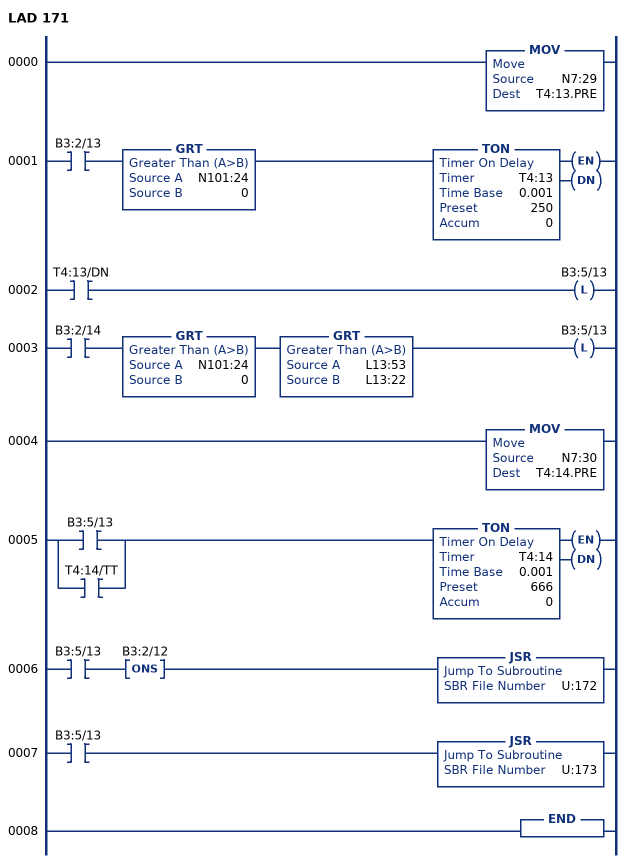
% Rung: 0 %
SOR MOV N7:29 T4:13.PRE EOR
% Rung: 1 %
SOR XIC B3:2/13 GRT N101:24 0 TON T4:13 0.001 250 0 EOR
% Rung: 2 %
SOR XIC T4:13/DN OTL B3:5/13 EOR
% Rung: 3 %
SOR XIC B3:2/14 GRT N101:24 0 GRT L13:53 L13:22 OTL B3:5/13 EOR
% Rung: 4 %
SOR MOV N7:30 T4:14.PRE EOR
% Rung: 5 %
SOR BST XIC B3:5/13 NXB XIC T4:14/TT BND TON T4:14 0.001 666 0 EOR
% Rung: 6 %
SOR XIC B3:5/13 ONS B3:2/12 JSR U:172 EOR
% Rung: 7 %
SOR XIC B3:5/13 JSR U:173 EOR
% Rung: 8 %
SOR END EOR

LADDER 172
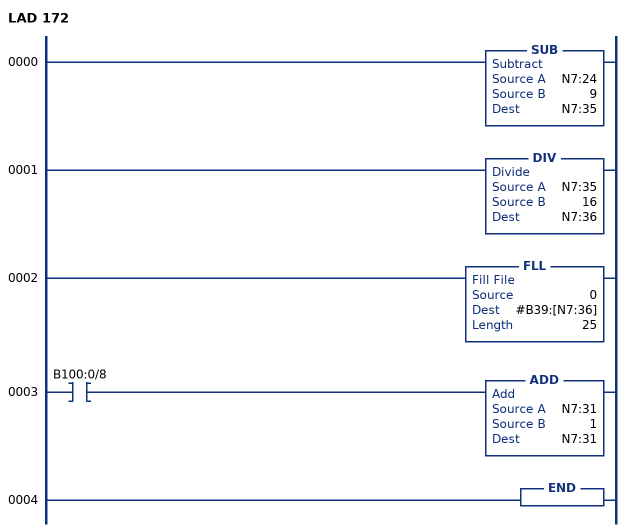
% Rung: 0 %
SOR SUB N7:24 9 N7:35 EOR
% Rung: 1 %
SOR DIV N7:35 16 N7:36 EOR
% Rung: 2 %
SOR FLL 0 #B39:[N7:36] 25 EOR
% Rung: 3 %
SOR XIC B100:0/8 ADD N7:31 1 N7:31 EOR
% Rung: 4 %
SOR END EOR

LADDER 173
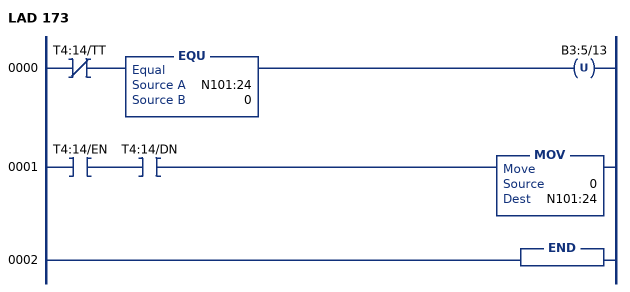
% Rung: 0 %
SOR XIO T4:14/TT EQU N101:24 0 OTU B3:5/13 EOR
% Rung: 1 %
SOR XIC T4:14/EN XIC T4:14/DN MOV 0 N101:24 EOR
% Rung: 2 %
SOR END EOR

LADDER 174
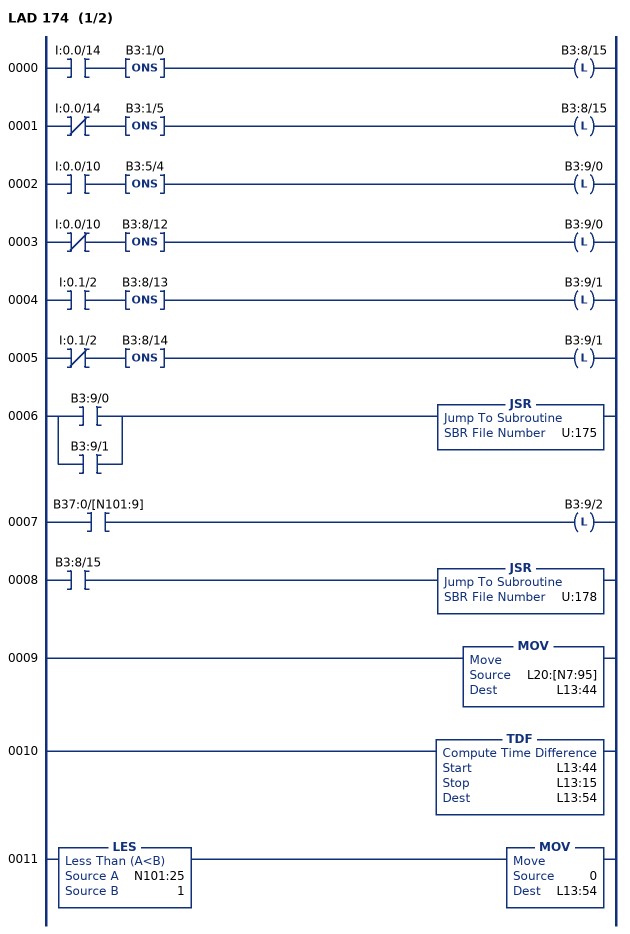
% Rung: 0 %
SOR XIC I:0.0/14 ONS B3:1/0 OTL B3:8/15 EOR
% Rung: 1 %
SOR XIO I:0.0/14 ONS B3:1/5 OTL B3:8/15 EOR
% Rung: 2 %
SOR XIC I:0.0/10 ONS B3:5/4 OTL B3:9/0 EOR
% Rung: 3 %
SOR XIO I:0.0/10 ONS B3:8/12 OTL B3:9/0 EOR
% Rung: 4 %
SOR XIC I:0.1/2 ONS B3:8/13 OTL B3:9/1 EOR
% Rung: 5 %
SOR XIO I:0.1/2 ONS B3:8/14 OTL B3:9/1 EOR
% Rung: 6 %
SOR BST XIC B3:9/0 NXB XIC B3:9/1 BND JSR U:175 EOR
% Rung: 7 %
SOR XIC B37:0/[N101:9] OTL B3:9/2 EOR
% Rung: 8 %
SOR XIC B3:8/15 JSR U:178 EOR
% Rung: 9 %
SOR MOV L20:[N7:95] L13:44 EOR
% Rung: 10 %
SOR TDF L13:44 L13:15 L13:54 EOR
% Rung: 11 %
SOR LES N101:25 1 MOV 0 L13:54 EOR

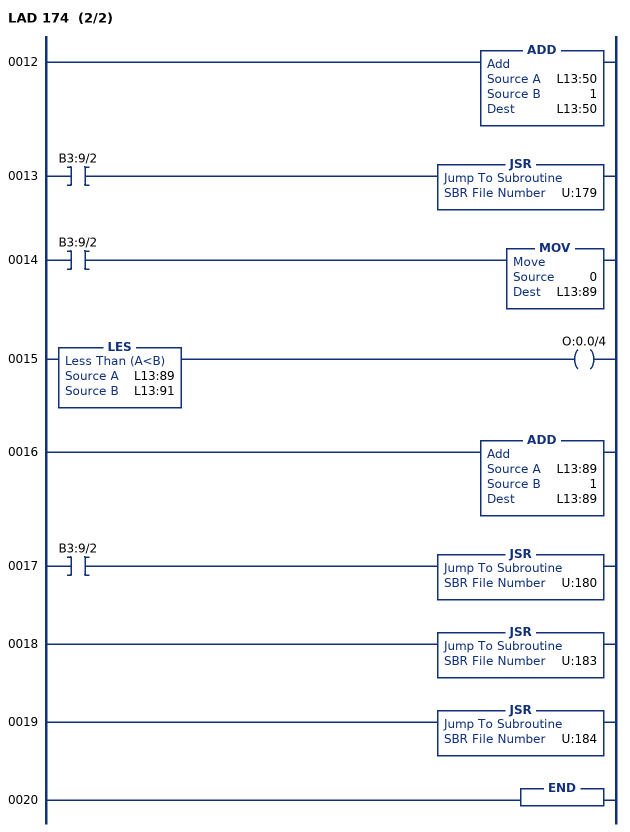
% Rung: 12 %
SOR ADD L13:50 1 L13:50 EOR
% Rung: 13 %
SOR XIC B3:9/2 JSR U:179 EOR
% Rung: 14 %
SOR XIC B3:9/2 MOV 0 L13:89 EOR
% Rung: 15 %
SOR LES L13:89 L13:91 OTE O:0.0/4 EOR
% Rung: 16 %
SOR ADD L13:89 1 L13:89 EOR
% Rung: 17 %
SOR XIC B3:9/2 JSR U:180 EOR
% Rung: 18 %
SOR JSR U:183 EOR
% Rung: 19 %
SOR JSR U:184 EOR
% Rung: 20 %
SOR END EOR

LADDER 175
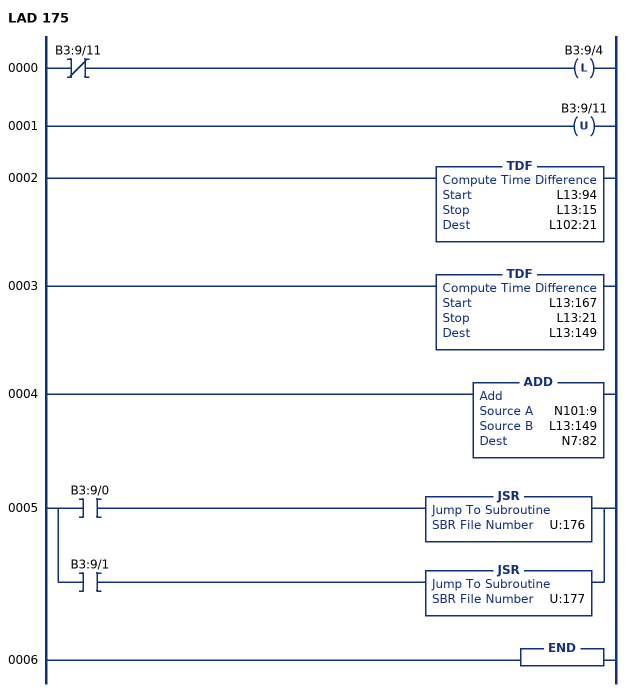
% Rung: 0 %
SOR XIO B3:9/11 OTL B3:9/4 EOR
% Rung: 1 %
SOR OTU B3:9/11 EOR
% Rung: 2 %
SOR TDF L13:94 L13:15 L102:21 EOR
% Rung: 3 %
SOR TDF L13:167 L13:21 L13:149 EOR
% Rung: 4 %
SOR ADD N101:9 L13:149 N7:82 EOR
% Rung: 5 %
SOR BST XIC B3:9/0 JSR U:176 NXB XIC B3:9/1 JSR U:177 BND EOR
% Rung: 6 %
SOR END EOR

LADDER 176
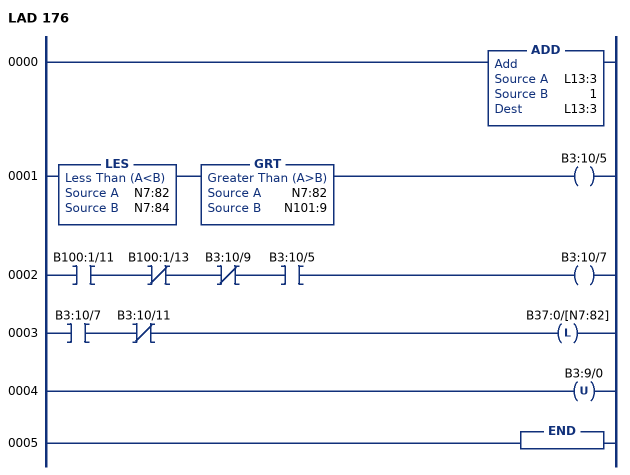
% Rung: 0 %
SOR ADD L13:3 1 L13:3 EOR
% Rung: 1 %
SOR LES N7:82 N7:84 GRT N7:82 N101:9 OTE B3:10/5 EOR
% Rung: 2 %
SOR XIC B100:1/11 XIO B100:1/13 XIO B3:10/9 XIC B3:10/5 OTE B3:10/7 EOR
% Rung: 3 %
SOR XIC B3:10/7 XIO B3:10/11 OTL B37:0/[N7:82] EOR
% Rung: 4 %
SOR OTU B3:9/0 EOR
% Rung: 5 %
SOR END EOR

LADDER 177
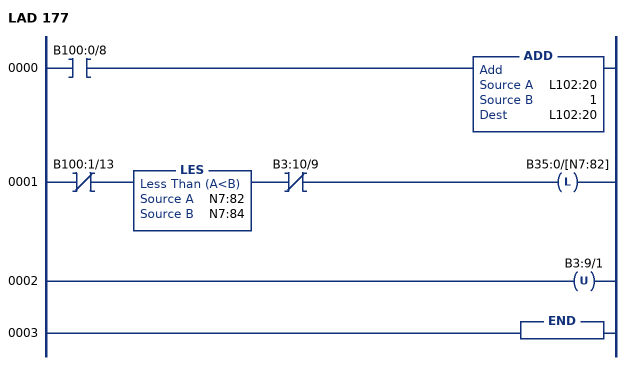
% Rung: 0 %
SOR XIC B100:0/8 ADD L102:20 1 L102:20 EOR
% Rung: 1 %
SOR XIO B100:1/13 LES N7:82 N7:84 XIO B3:10/9 OTL B35:0/[N7:82] EOR
% Rung: 2 %
SOR OTU B3:9/1 EOR
% Rung: 3 %
SOR END EOR

LADDER 178
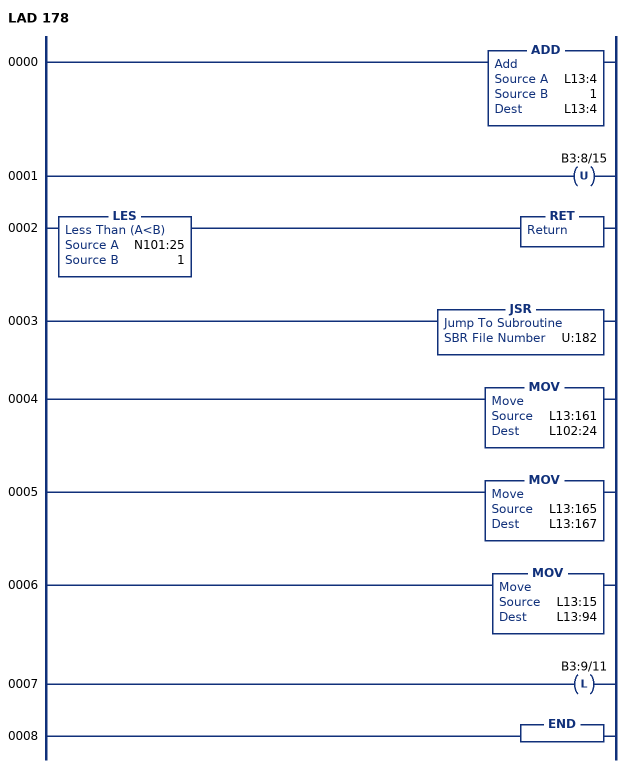
% Rung: 0 %
SOR ADD L13:4 1 L13:4 EOR
% Rung: 1 %
SOR OTU B3:8/15 EOR
% Rung: 2 %
SOR LES N101:25 1 RET EOR
% Rung: 3 %
SOR JSR U:182 EOR
% Rung: 4 %
SOR MOV L13:161 L102:24 EOR
% Rung: 5 %
SOR MOV L13:165 L13:167 EOR
% Rung: 6 %
SOR MOV L13:15 L13:94 EOR
% Rung: 7 %
SOR OTL B3:9/11 EOR
% Rung: 8 %
SOR END EOR

LADDER 179
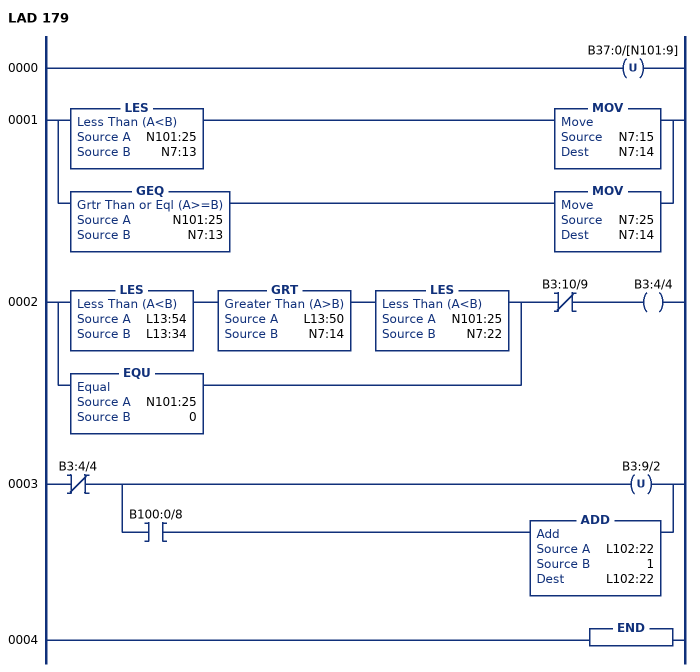
% Rung: 0 %
SOR OTU B37:0/[N101:9] EOR
% Rung: 1 %
SOR BST LES N101:25 N7:13 MOV N7:15 N7:14 NXB GEQ N101:25 N7:13 MOV N7:25 N7:14 BND EOR
% Rung: 2 %
SOR BST LES L13:54 L13:34 GRT L13:50 N7:14 LES N101:25 N7:22 NXB EQU N101:25 0 BND XIO B3:10/9 OTE B3:4/4 EOR
% Rung: 3 %
SOR XIO B3:4/4 BST OTU B3:9/2 NXB XIC B100:0/8 ADD L102:22 1 L102:22 BND EOR
% Rung: 4 %
SOR END EOR

LADDER 180
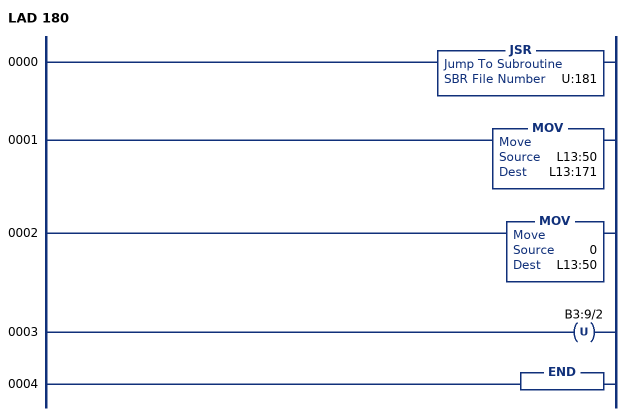
% Rung: 0 %
SOR JSR U:181 EOR
% Rung: 1 %
SOR MOV L13:50 L13:171 EOR
% Rung: 2 %
SOR MOV 0 L13:50 EOR
% Rung: 3 %
SOR OTU B3:9/2 EOR
% Rung: 4 %
SOR END EOR

LADDER 181
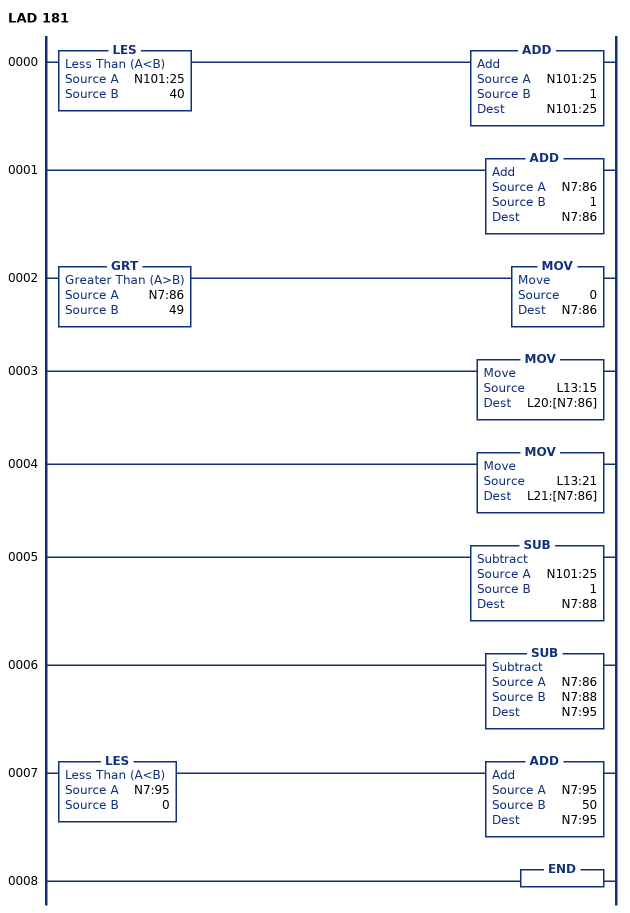
% Rung: 0 %
SOR LES N101:25 40 ADD N101:25 1 N101:25 EOR
% Rung: 1 %
SOR ADD N7:86 1 N7:86 EOR
% Rung: 2 %
SOR GRT N7:86 49 MOV 0 N7:86 EOR
% Rung: 3 %
SOR MOV L13:15 L20:[N7:86] EOR
% Rung: 4 %
SOR MOV L13:21 L21:[N7:86] EOR
% Rung: 5 %
SOR SUB N101:25 1 N7:88 EOR
% Rung: 6 %
SOR SUB N7:86 N7:88 N7:95 EOR
% Rung: 7 %
SOR LES N7:95 0 ADD N7:95 50 N7:95 EOR
% Rung: 8 %
SOR END EOR

LADDER 182
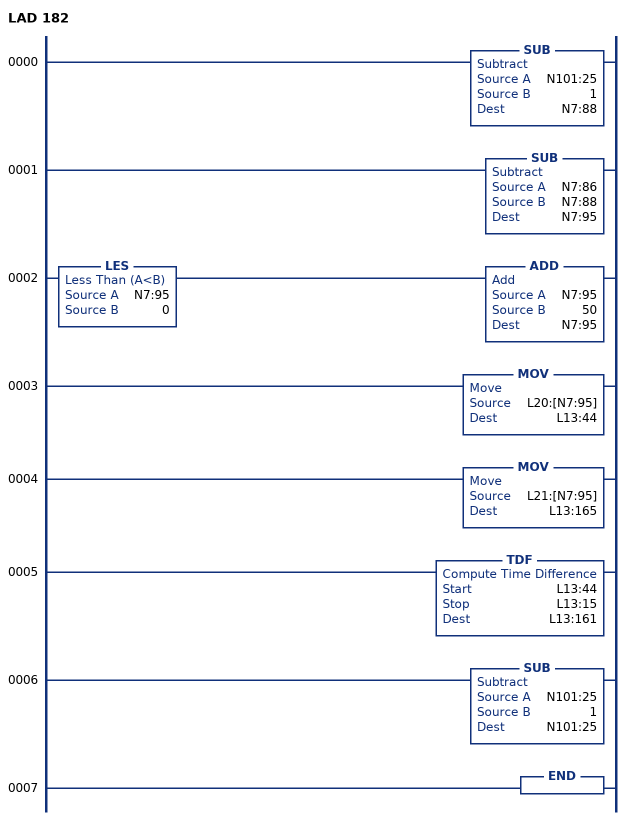
% Rung: 0 %
SOR SUB N101:25 1 N7:88 EOR
% Rung: 1 %
SOR SUB N7:86 N7:88 N7:95 EOR
% Rung: 2 %
SOR LES N7:95 0 ADD N7:95 50 N7:95 EOR
% Rung: 3 %
SOR MOV L20:[N7:95] L13:44 EOR
% Rung: 4 %
SOR MOV L21:[N7:95] L13:165 EOR
% Rung: 5 %
SOR TDF L13:44 L13:15 L13:161 EOR
% Rung: 6 %
SOR SUB N101:25 1 N101:25 EOR
% Rung: 7 %
SOR END EOR

LADDER 183
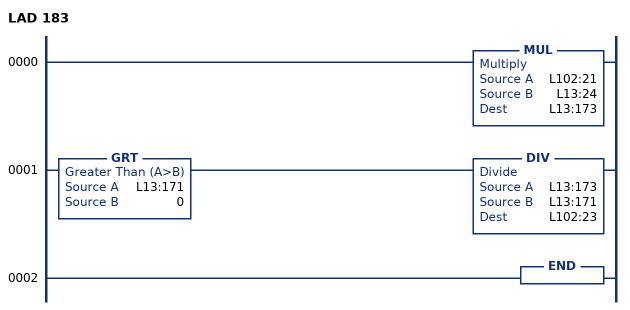
% Rung: 0 %
SOR MUL L102:21 L13:24 L13:173 EOR
% Rung: 1 %
SOR GRT L13:171 0 DIV L13:173 L13:171 L102:23 EOR
% Rung: 2 %
SOR END EOR

LADDER 184
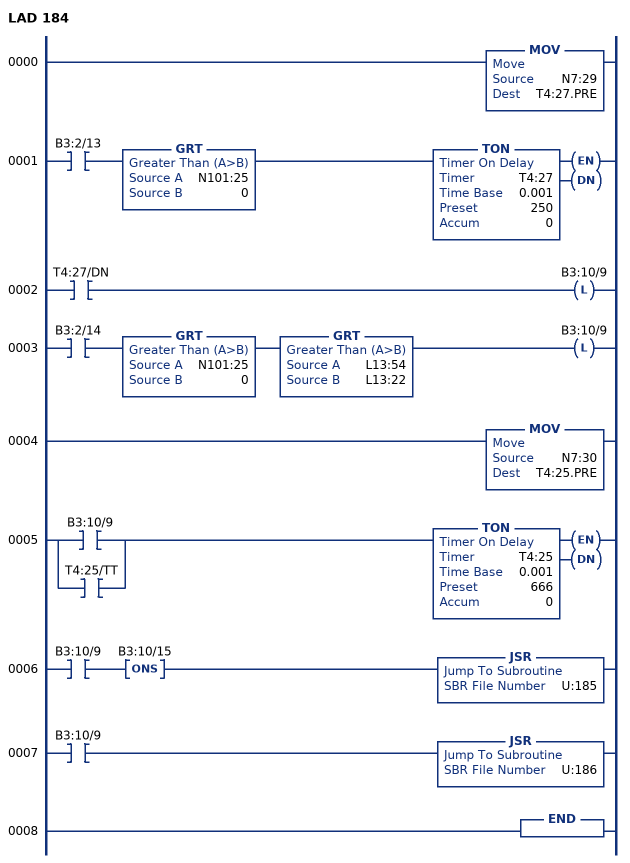
% Rung: 0 %
SOR MOV N7:29 T4:27.PRE EOR
% Rung: 1 %
SOR XIC B3:2/13 GRT N101:25 0 TON T4:27 0.001 250 0 EOR
% Rung: 2 %
SOR XIC T4:27/DN OTL B3:10/9 EOR
% Rung: 3 %
SOR XIC B3:2/14 GRT N101:25 0 GRT L13:54 L13:22 OTL B3:10/9 EOR
% Rung: 4 %
SOR MOV N7:30 T4:25.PRE EOR
% Rung: 5 %
SOR BST XIC B3:10/9 NXB XIC T4:25/TT BND TON T4:25 0.001 666 0 EOR
% Rung: 6 %
SOR XIC B3:10/9 ONS B3:10/15 JSR U:185 EOR
% Rung: 7 %
SOR XIC B3:10/9 JSR U:186 EOR
% Rung: 8 %
SOR END EOR

LADDER 185
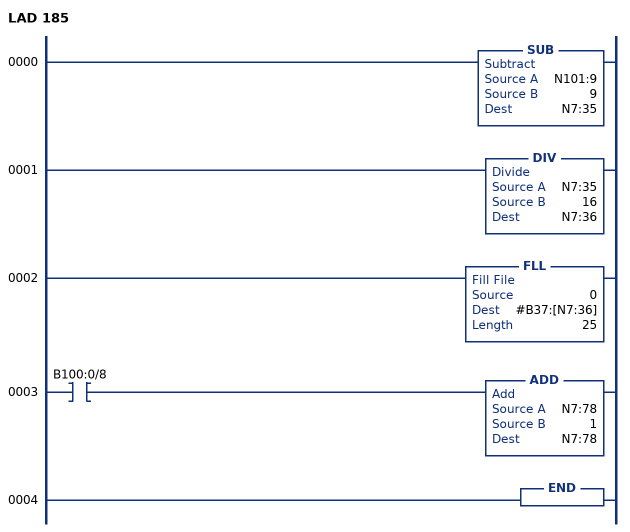
% Rung: 0 %
SOR SUB N101:9 9 N7:35 EOR
% Rung: 1 %
SOR DIV N7:35 16 N7:36 EOR
% Rung: 2 %
SOR FLL 0 #B37:[N7:36] 25 EOR
% Rung: 3 %
SOR XIC B100:0/8 ADD N7:78 1 N7:78 EOR
% Rung: 4 %
SOR END EOR

LADDER 186
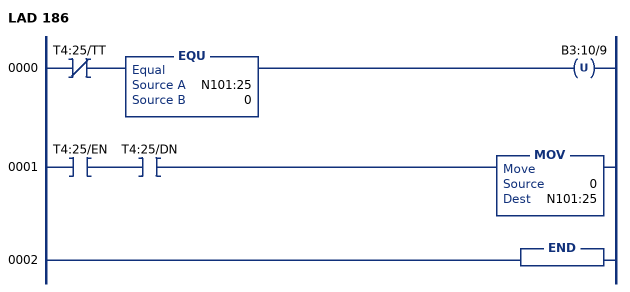
% Rung: 0 %
SOR XIO T4:25/TT EQU N101:25 0 OTU B3:10/9 EOR
% Rung: 1 %
SOR XIC T4:25/EN XIC T4:25/DN MOV 0 N101:25 EOR
% Rung: 2 %
SOR END EOR

LADDER 187
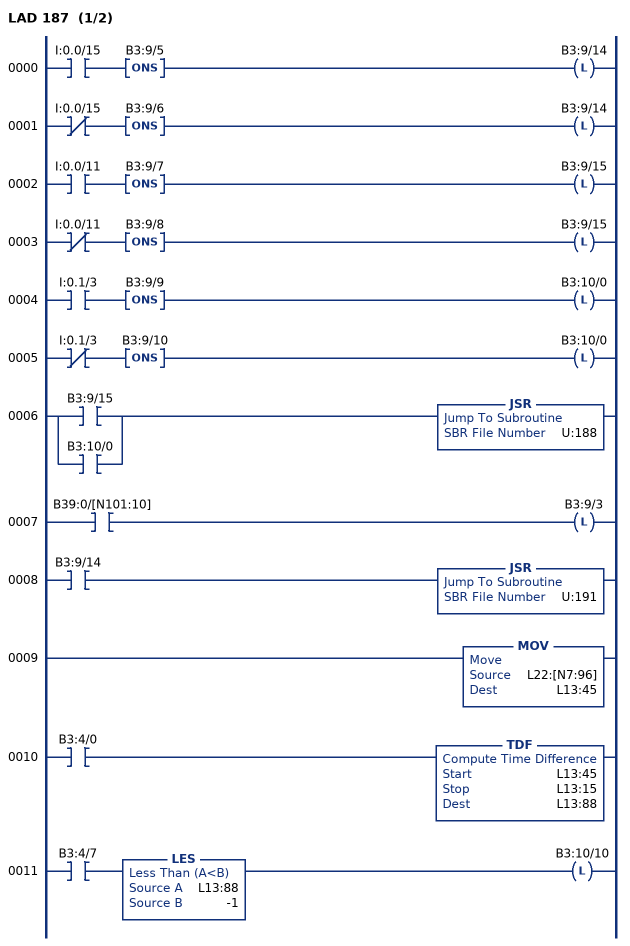
% Rung: 0 %
SOR XIC I:0.0/15 ONS B3:9/5 OTL B3:9/14 EOR
% Rung: 1 %
SOR XIO I:0.0/15 ONS B3:9/6 OTL B3:9/14 EOR
% Rung: 2 %
SOR XIC I:0.0/11 ONS B3:9/7 OTL B3:9/15 EOR
% Rung: 3 %
SOR XIO I:0.0/11 ONS B3:9/8 OTL B3:9/15 EOR
% Rung: 4 %
SOR XIC I:0.1/3 ONS B3:9/9 OTL B3:10/0 EOR
% Rung: 5 %
SOR XIO I:0.1/3 ONS B3:9/10 OTL B3:10/0 EOR
% Rung: 6 %
SOR BST XIC B3:9/15 NXB XIC B3:10/0 BND JSR U:188 EOR
% Rung: 7 %
SOR XIC B39:0/[N101:10] OTL B3:9/3 EOR
% Rung: 8 %
SOR XIC B3:9/14 JSR U:191 EOR
% Rung: 9 %
SOR MOV L22:[N7:96] L13:45 EOR
% Rung: 10 %
SOR XIC B3:4/0 TDF L13:45 L13:15 L13:88 EOR
% Rung: 11 %
SOR XIC B3:4/7 LES L13:88 -1 OTL B3:10/10 EOR

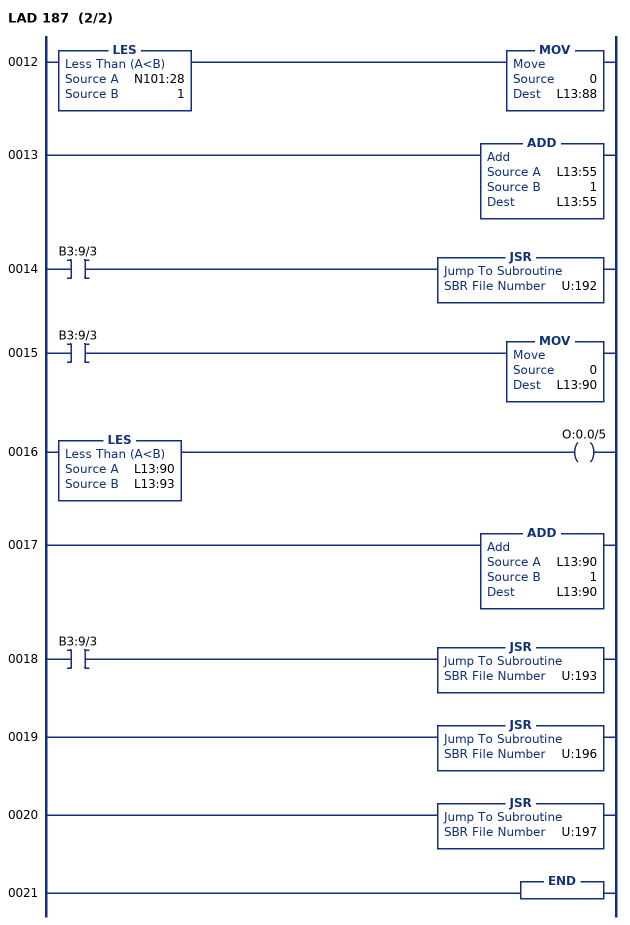
% Rung: 12 %
SOR LES N101:28 1 MOV 0 L13:88 EOR
% Rung: 13 %
SOR ADD L13:55 1 L13:55 EOR
% Rung: 14 %
SOR XIC B3:9/3 JSR U:192 EOR
% Rung: 15 %
SOR XIC B3:9/3 MOV 0 L13:90 EOR
% Rung: 16 %
SOR LES L13:90 L13:93 OTE O:0.0/5 EOR
% Rung: 17 %
SOR ADD L13:90 1 L13:90 EOR
% Rung: 18 %
SOR XIC B3:9/3 JSR U:193 EOR
% Rung: 19 %
SOR JSR U:196 EOR
% Rung: 20 %
SOR JSR U:197 EOR
% Rung: 21 %
SOR END EOR

LADDER 188
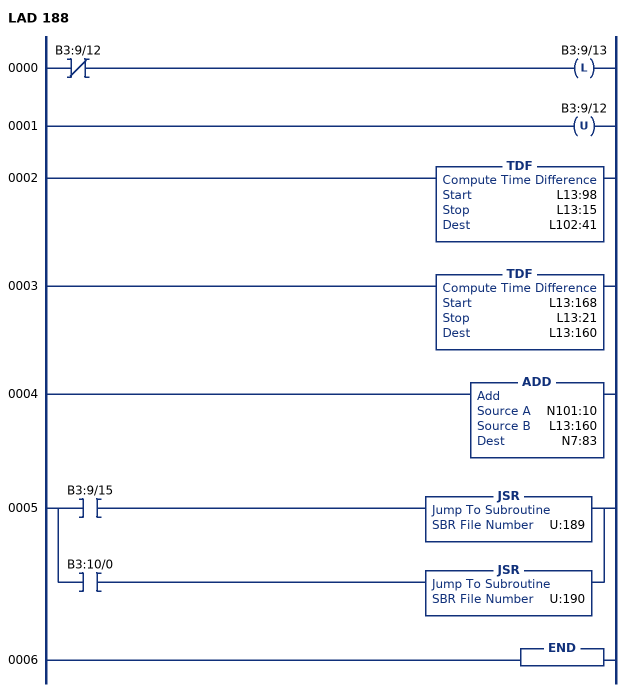
% Rung: 0 %
SOR XIO B3:9/12 OTL B3:9/13 EOR
% Rung: 1 %
SOR OTU B3:9/12 EOR
% Rung: 2 %
SOR TDF L13:98 L13:15 L102:41 EOR
% Rung: 3 %
SOR TDF L13:168 L13:21 L13:160 EOR
% Rung: 4 %
SOR ADD N101:10 L13:160 N7:83 EOR
% Rung: 5 %
SOR BST XIC B3:9/15 JSR U:189 NXB XIC B3:10/0 JSR U:190 BND EOR
% Rung: 6 %
SOR END EOR

LADDER 189
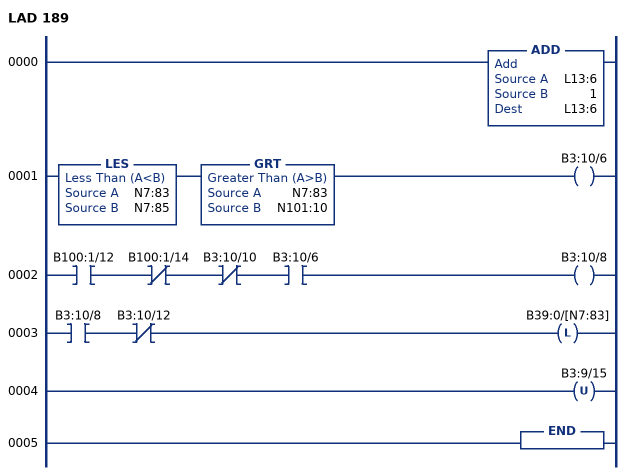
% Rung: 0 %
SOR ADD L13:6 1 L13:6 EOR
% Rung: 1 %
SOR LES N7:83 N7:85 GRT N7:83 N101:10 OTE B3:10/6 EOR
% Rung: 2 %
SOR XIC B100:1/12 XIO B100:1/14 XIO B3:10/10 XIC B3:10/6 OTE B3:10/8 EOR
% Rung: 3 %
SOR XIC B3:10/8 XIO B3:10/12 OTL B39:0/[N7:83] EOR
% Rung: 4 %
SOR OTU B3:9/15 EOR
% Rung: 5 %
SOR END EOR

LADDER 190
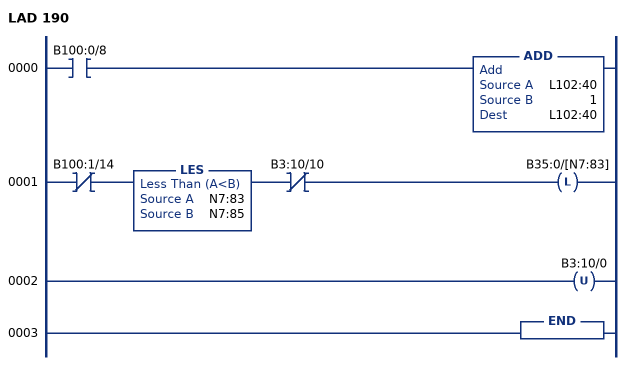
% Rung: 0 %
SOR XIC B100:0/8 ADD L102:40 1 L102:40 EOR
% Rung: 1 %
SOR XIO B100:1/14 LES N7:83 N7:85 XIO B3:10/10 OTL B35:0/[N7:83] EOR
% Rung: 2 %
SOR OTU B3:10/0 EOR
% Rung: 3 %
SOR END EOR

LADDER 191
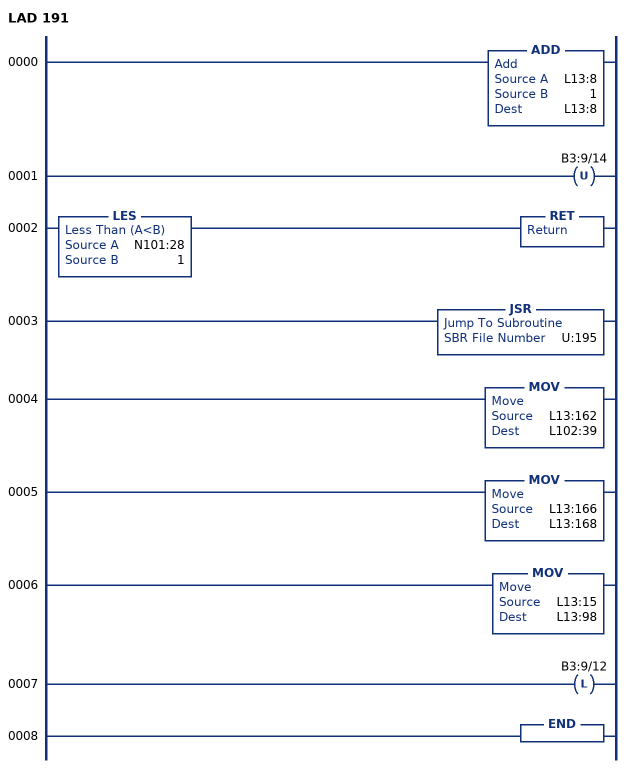
% Rung: 0 %
SOR ADD L13:8 1 L13:8 EOR
% Rung: 1 %
SOR OTU B3:9/14 EOR
% Rung: 2 %
SOR LES N101:28 1 RET EOR
% Rung: 3 %
SOR JSR U:195 EOR
% Rung: 4 %
SOR MOV L13:162 L102:39 EOR
% Rung: 5 %
SOR MOV L13:166 L13:168 EOR
% Rung: 6 %
SOR MOV L13:15 L13:98 EOR
% Rung: 7 %
SOR OTL B3:9/12 EOR
% Rung: 8 %
SOR END EOR

LADDER 192
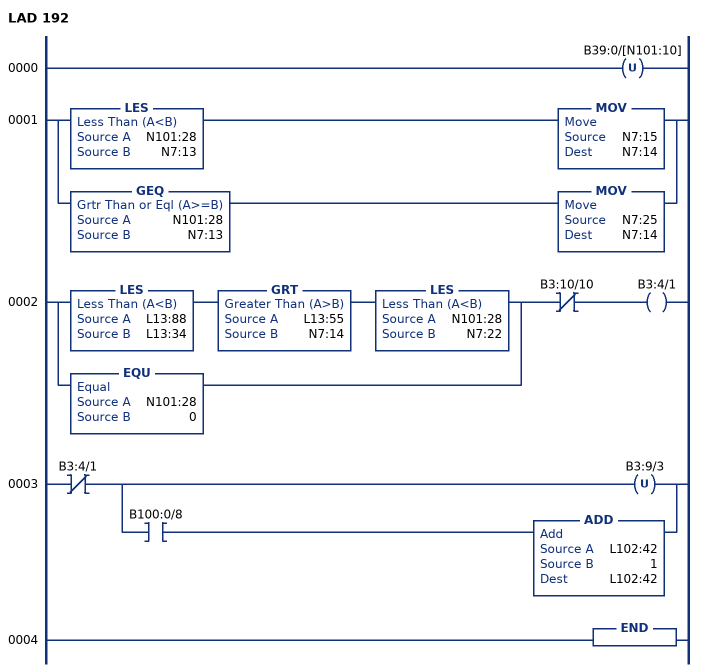
% Rung: 0 %
SOR OTU B39:0/[N101:10] EOR
% Rung: 1 %
SOR BST LES N101:28 N7:13 MOV N7:15 N7:14 NXB GEQ N101:28 N7:13 MOV N7:25 N7:14 BND EOR
% Rung: 2 %
SOR BST LES L13:88 L13:34 GRT L13:55 N7:14 LES N101:28 N7:22 NXB EQU N101:28 0 BND XIO B3:10/10 OTE B3:4/1 EOR
% Rung: 3 %
SOR XIO B3:4/1 BST OTU B3:9/3 NXB XIC B100:0/8 ADD L102:42 1 L102:42 BND EOR
% Rung: 4 %
SOR END EOR

LADDER 193
